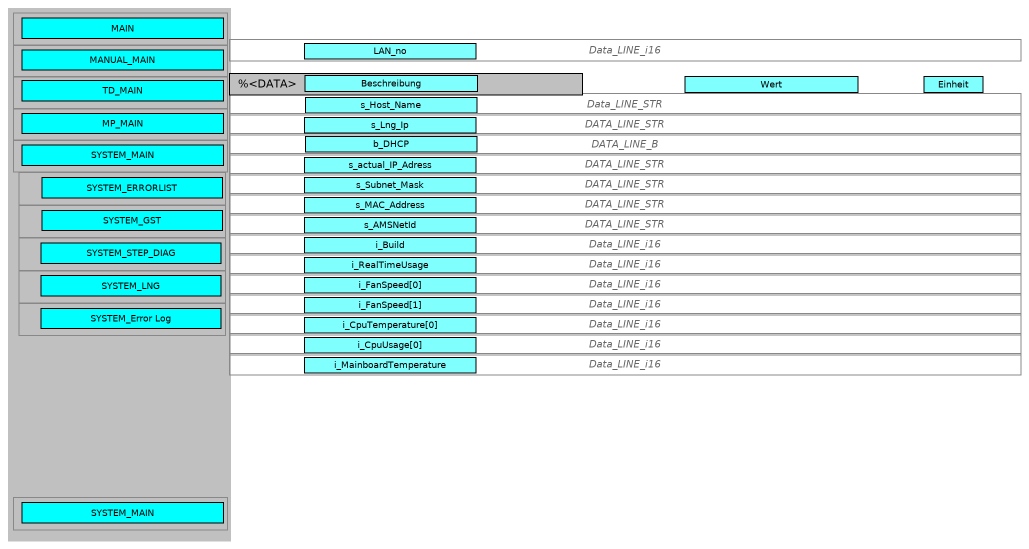
[picture p157: SYSTEM_MAIN (HMI screen)]
embedded screen at (3,115)-(226,648): M0003_System
embedded screen at (224,200)-(1016,222): Data_LINE_STR
embedded screen at (224,240)-(1016,262): DATA_LINE_B
rectangle at (300,204)-(472,220): text "s_Host_Name"; invisible if TRUE
rectangle at (300,243)-(472,259): text "b_DHCP"; invisible if TRUE
embedded screen at (224,260)-(1016,282): DATA_LINE_STR
rectangle at (299,264)-(471,280): text "s_actual_IP_Adress"; invisible if TRUE
embedded screen at (224,280)-(1016,302): DATA_LINE_STR
rectangle at (299,284)-(471,300): text "s_Subnet_Mask"; invisible if TRUE
embedded screen at (224,300)-(1016,322): DATA_LINE_STR
rectangle at (299,304)-(471,320): text "s_MAC_Address"; invisible if TRUE
embedded screen at (224,320)-(1016,342): DATA_LINE_STR
rectangle at (299,324)-(471,340): text "s_AMSNetId"; invisible if TRUE
embedded screen at (224,340)-(1016,362): Data_LINE_i16
rectangle at (299,344)-(471,360): text "i_Build"; invisible if TRUE
embedded screen at (224,360)-(1016,382): Data_LINE_i16
rectangle at (299,364)-(471,380): text "i_RealTimeUsage"; invisible if TRUE
embedded screen at (224,380)-(1016,402): Data_LINE_i16
rectangle at (299,384)-(471,400): text "i_FanSpeed[0]"; invisible if TRUE
embedded screen at (224,400)-(1016,422): Data_LINE_i16
rectangle at (299,404)-(471,420): text "i_FanSpeed[1]"; invisible if TRUE
embedded screen at (224,420)-(1016,442): Data_LINE_i16
rectangle at (299,424)-(471,440): text "i_CpuTemperature[0]"; invisible if TRUE
embedded screen at (224,440)-(1016,462): Data_LINE_i16
rectangle at (299,444)-(471,460): text "i_CpuUsage[0]"; invisible if TRUE
embedded screen at (224,460)-(1016,482): Data_LINE_i16
rectangle at (299,464)-(471,480): text "i_MainboardTemperature"; invisible if TRUE
embedded screen at (224,180)-(978,202): DATA_HEADER
embedded screen at (224,220)-(1016,242): DATA_LINE_STR
rectangle at (299,224)-(471,240): text "s_Lng_Ip"; invisible if TRUE
embedded screen at (224,146)-(1016,168): Data_LINE_i16
rectangle at (299,150)-(471,166): text "LAN_no"; invisible if TRUE
*)

(* Visualisation 04_System/SYSTEM_STEP_DIAG
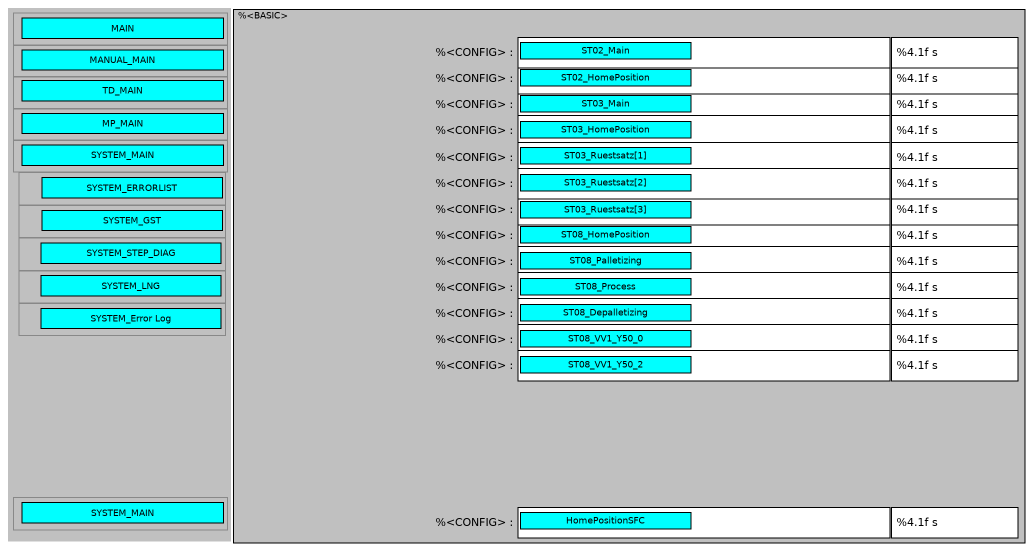
rectangle at (228,115)-(1020,649): text "%<BASIC>"; shows 'Prozess-Schrittketten'
embedded screen at (3,114)-(226,647): M0003_System
embedded screen at (282,195)-(1013,226): ZLIB_SFC_STATE
embedded screen at (282,221)-(1013,252): ZLIB_SFC_STATE
embedded screen at (282,326)-(1013,357): ZLIB_SFC_STATE
embedded screen at (282,352)-(1013,383): ZLIB_SFC_STATE
embedded screen at (282,378)-(1013,409): ZLIB_SFC_STATE
embedded screen at (282,404)-(1013,435): ZLIB_SFC_STATE
embedded screen at (282,430)-(1013,461): ZLIB_SFC_STATE
embedded screen at (282,456)-(1013,487): ZLIB_SFC_STATE
embedded screen at (282,300)-(1013,331): ZLIB_SFC_STATE
embedded screen at (282,613)-(1013,644): ZLIB_SFC_STATE
embedded screen at (282,169)-(1013,200): ZLIB_SFC_STATE
embedded screen at (282,143)-(1013,174): ZLIB_SFC_STATE
rectangle at (515,148)-(686,165): text "ST02_Main"; invisible if TRUE
rectangle at (515,175)-(686,192): text "ST02_HomePosition"; invisible if TRUE
rectangle at (515,201)-(686,218): text "ST03_Main"; invisible if TRUE
rectangle at (515,227)-(686,244): text "ST03_HomePosition"; invisible if TRUE
rectangle at (515,332)-(686,349): text "ST08_HomePosition"; invisible if TRUE
rectangle at (515,358)-(686,375): text "ST08_Palletizing"; invisible if TRUE
rectangle at (515,384)-(686,401): text "ST08_Process"; invisible if TRUE
rectangle at (515,410)-(686,427): text "ST08_Depalletizing"; invisible if TRUE
rectangle at (515,436)-(686,453): text "ST08_VV1_Y50_0"; invisible if TRUE
rectangle at (515,462)-(686,479): text "ST08_VV1_Y50_2"; invisible if TRUE
rectangle at (515,307)-(686,324): text "ST03_Ruestsatz[3]"; invisible if TRUE
rectangle at (515,618)-(686,635): text "HomePositionSFC"; invisible if TRUE
embedded screen at (282,248)-(1013,279): ZLIB_SFC_STATE
embedded screen at (282,274)-(1013,305): ZLIB_SFC_STATE
rectangle at (515,253)-(686,270): text "ST03_Ruestsatz[1]"; invisible if TRUE
rectangle at (515,280)-(686,297): text "ST03_Ruestsatz[2]"; invisible if TRUE
*)

(* Visualisation 02_TypeData/TD_01_EDIT
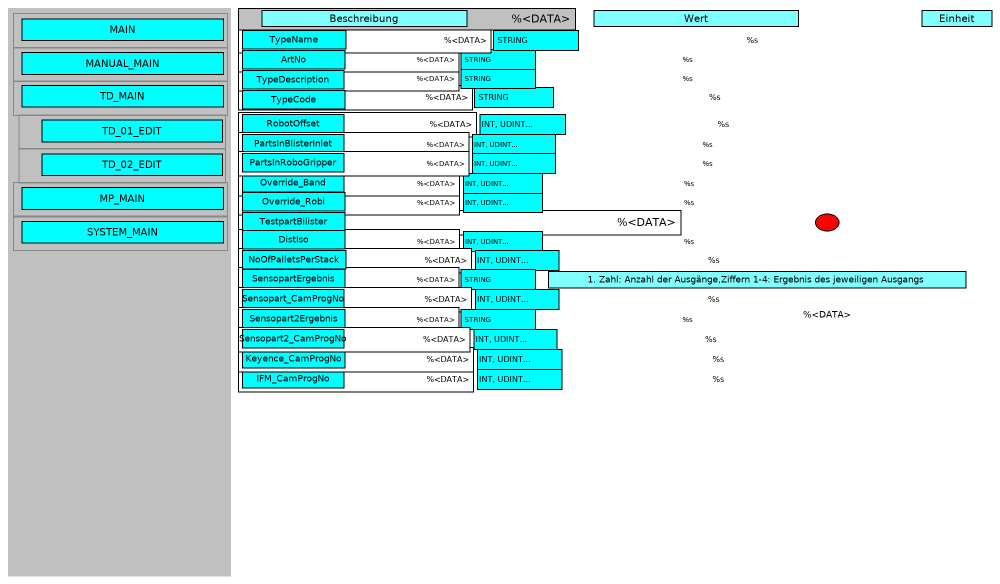
embedded screen at (3,115)-(226,683): M0003_TD
rectangle at (796,407)-(1009,436): text "%<DATA>"; shows 'Info_01'; invisible if gTypeCode<>4991 AND gTypeCode <>312
embedded screen at (233,317)-(834,342): Data_BOOL
embedded screen at (233,192)-(870,217): Data_STRING
embedded screen at (233,297)-(834,322): Data_DEZIMAL
embedded screen at (233,278)-(834,303): Data_DEZIMAL
embedded screen at (233,173)-(834,198): Data_STRING
embedded screen at (233,154)-(834,179): Data_STRING
embedded screen at (233,135)-(921,160): Data_STRING
embedded screen at (233,336)-(834,361): Data_DEZIMAL
embedded screen at (233,355)-(866,380): Data_DEZIMAL
embedded screen at (233,374)-(834,399): Data_STRING
rectangle at (237,137)-(341,156): text "TypeName"; invisible if TRUE
rectangle at (237,157)-(340,176): text "ArtNo"; invisible if TRUE
rectangle at (237,177)-(339,196): text "TypeDescription"; invisible if TRUE
rectangle at (237,197)-(340,216): text "TypeCode"; invisible if TRUE
rectangle at (237,280)-(339,299): text "Override_Band"; invisible if TRUE
rectangle at (237,299)-(340,318): text "Override_Robi"; invisible if TRUE
rectangle at (237,319)-(340,338): text "TestpartBilister"; invisible if TRUE
rectangle at (237,337)-(340,356): text "DistIso"; invisible if TRUE
rectangle at (237,376)-(340,395): text "SensopartErgebnis"; invisible if TRUE
rectangle at (237,357)-(341,376): text "NoOfPalletsPerStack"; invisible if TRUE
rectangle at (543,378)-(961,395): text "1. Zahl: Anzahl der Ausgänge,Ziffern 1-4: Ergebnis des jeweiligen Ausgangs"; invisible if TRUE
embedded screen at (233,219)-(879,244): Data_DEZIMAL
rectangle at (237,221)-(339,240): text "RobotOffset"; invisible if TRUE
embedded screen at (233,239)-(859,264): Data_DEZIMAL
rectangle at (237,241)-(339,260): text "PartsInBlisterInlet"; invisible if TRUE
embedded screen at (233,474)-(872,499): Data_DEZIMAL
rectangle at (237,476)-(339,495): text "IFM_CamProgNo"; invisible if TRUE
embedded screen at (233,394)-(866,419): Data_DEZIMAL
rectangle at (237,396)-(339,415): text "Sensopart_CamProgNo"; invisible if TRUE
embedded screen at (233,258)-(859,283): Data_DEZIMAL
rectangle at (237,260)-(339,279): text "PartsInRoboGripper"; invisible if TRUE
embedded screen at (233,115)-(987,137): DATA_HEADER_BEER
embedded screen at (233,454)-(872,479): Data_DEZIMAL
rectangle at (237,456)-(340,475): text "Keyence_CamProgNo"; invisible if TRUE
embedded screen at (233,414)-(834,439): Data_STRING
rectangle at (237,416)-(340,435): text "Sensopart2Ergebnis"; invisible if TRUE
embedded screen at (233,434)-(862,459): Data_DEZIMAL
rectangle at (237,436)-(339,455): text "Sensopart2_CamProgNo"; invisible if TRUE
*)

(* Visualisation 02_TypeData/TD_02_EDIT
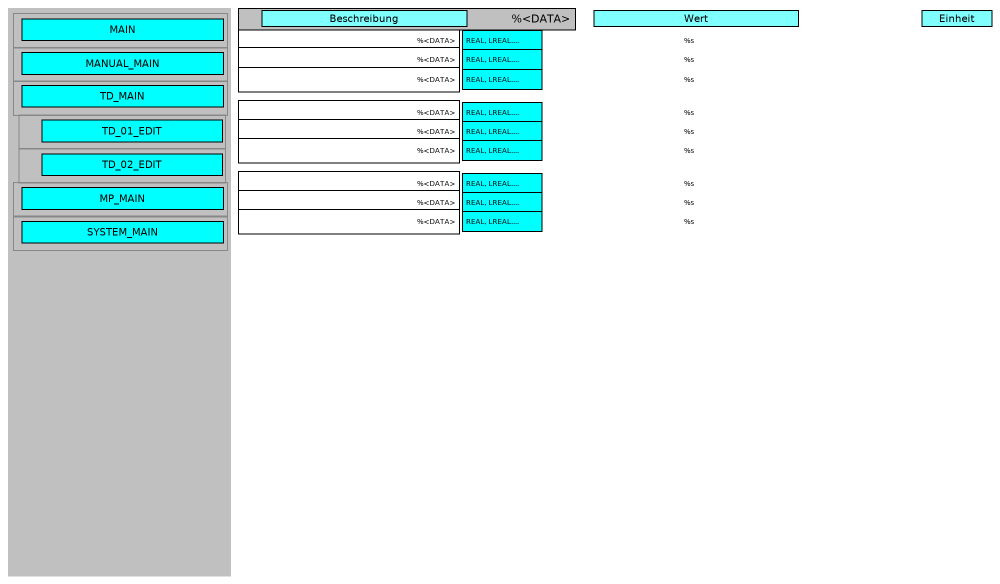
embedded screen at (3,115)-(226,683): M0003_TD
embedded screen at (233,135)-(834,160): Data_DEZIMAL_REAL
embedded screen at (233,154)-(834,179): Data_DEZIMAL_REAL
embedded screen at (233,174)-(834,199): Data_DEZIMAL_REAL
embedded screen at (233,207)-(834,232): Data_DEZIMAL_REAL
embedded screen at (233,226)-(834,251): Data_DEZIMAL_REAL
embedded screen at (233,245)-(834,270): Data_DEZIMAL_REAL
embedded screen at (233,115)-(987,137): DATA_HEADER_BEER
embedded screen at (233,278)-(834,303): Data_DEZIMAL_REAL
embedded screen at (233,297)-(834,322): Data_DEZIMAL_REAL
embedded screen at (233,316)-(834,341): Data_DEZIMAL_REAL
*)

(* Visualisation 02_TypeData/TD_MAIN
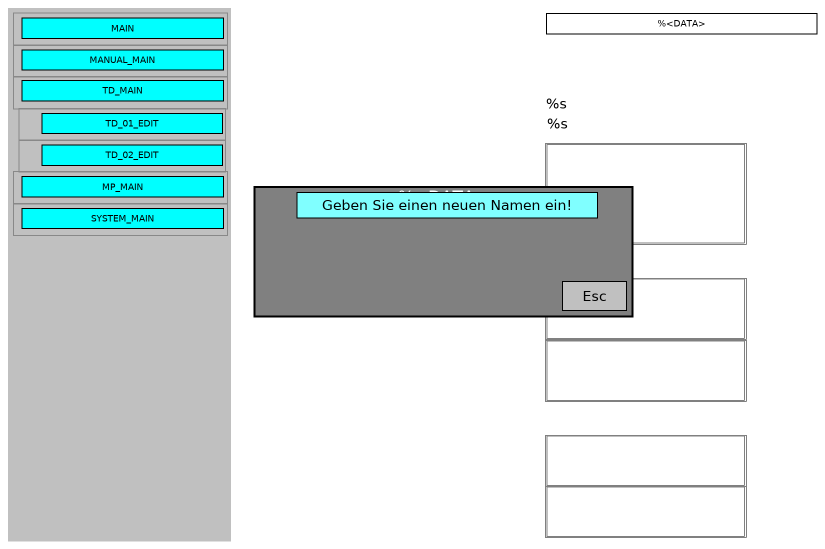
rectangle at (541,120)-(812,141): text "%<DATA>"; shows 'Filter'
embedded screen at (540,250)-(741,351): ZLIB_VISUBUTTON
embedded screen at (540,447)-(741,508): ZLIB_VISUBUTTON
embedded screen at (3,115)-(226,648): M0003_TD
embedded screen at (540,542)-(741,593): ZLIB_VISUBUTTON
embedded screen at (540,593)-(741,644): ZLIB_VISUBUTTON
embedded screen at (540,385)-(741,446): ZLIB_VISUBUTTON
embedded screen at (247,293)-(628,424): DIALOG_SAVE_AS
rectangle at (539,200)-(730,221): text "%s"; shows TDHandler.s_Typecode
rectangle at (540,220)-(731,241): text "%s"; shows TDHandler.s_Typedescription
2 elements of other kinds (tables, trends, ...) not read
*)

(* Visualisation zLibrary/ept/TEILEZAEHLER
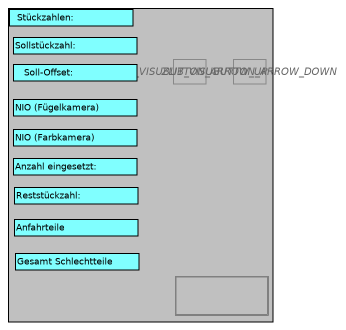
rectangle at (0,0)-(265,314): text "%<DATA>"; shows 'Parts'
rectangle at (10,23)-(157,48): text "%<DATA>"; shows 'PartsToProduce'
rectangle at (10,51)-(157,76): text "%<DATA>"; shows 'PartsToProduceOffset'
rectangle at (10,146)-(157,171): text "%<DATA>"; shows 'gPartsInserted'
rectangle at (10,176)-(157,201): text "%<DATA>"; shows 'PartsRemaining'
embedded screen at (165,51)-(198,76): ZLIB_VISUBUTTON_ARROW_UP
embedded screen at (225,51)-(258,76): ZLIB_VISUBUTTON_ARROW_DOWN
embedded screen at (167,268)-(260,307): ZLIB_VISUBUTTON_S18
rectangle at (10,116)-(157,141): text "%<DATA>"; shows 'gNokPartsColorCam'; invisible if gTypeCode<>5633 AND gTypeCode<>4991 AND gTypeCode <>312 AND gTypeCode <>322
rectangle at (10,86)-(157,111): text "%<DATA>"; shows 'gNokPartsWingCam'; invisible if gTypeCode<>4991 AND gTypeCode <>312
rectangle at (1,1)-(125,18): text "Stückzahlen:"; invisible if TRUE
rectangle at (5,29)-(129,46): text "Sollstückzahl:"; invisible if TRUE
rectangle at (5,56)-(129,73): text "Soll-Offset:"; invisible if TRUE
rectangle at (5,91)-(129,108): text "NIO (Fügelkamera)"; invisible if TRUE
rectangle at (5,121)-(129,138): text "NIO (Farbkamera)"; invisible if TRUE
rectangle at (5,150)-(129,167): text "Anzahl eingesetzt:"; invisible if TRUE
rectangle at (6,179)-(130,196): text "Reststückzahl:"; invisible if TRUE
rectangle at (10,207)-(166,232): text "%<DATA>"; shows 'Anfahrteile'
rectangle at (10,238)-(170,263): text "%<DATA>"; shows 'Gesamt Schlechtteile'
rectangle at (6,211)-(130,228): text "Anfahrteile"; invisible if TRUE
rectangle at (7,245)-(131,262): text "Gesamt Schlechtteile"; invisible if TRUE
9 elements of other kinds (tables, trends, ...) not read
*)

(* Visualisation zLibrary/MachineObjects/AnaIn/VANAIN
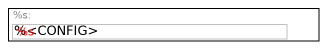
rectangle at (0,0)-(311,33): text "%s:"; shows $Object$.BitInName
rectangle at (0,12)-(281,33): text "%<CONFIG>"; shows $Object$.InstName
rectangle at (4,16)-(279,31): text "%s"; shows $Object$.ErrorString; invisible if NOT $Object$.ErrorPresent
1 elements of other kinds (tables, trends, ...) not read
*)

(* Visualisation zLibrary/MachineObjects/DigInOut/VBTN_SMAL
1 elements of other kinds (tables, trends, ...) not read
*)

(* Visualisation zLibrary/MachineObjects/DigIn/VDIGIN
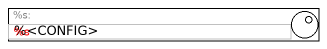
rectangle at (0,0)-(311,33): text "%s:"; shows $Object$.BitInName
rectangle at (0,12)-(281,33): text "%<CONFIG>"; shows $Object$.InstName
rectangle at (0,16)-(283,31): text "%s"; shows $Object$.ErrorString; invisible if NOT $Object$.ErrorPresent OR TRUE; alarm colour if $Object$.ErrorPresent
group at (283,3)-(310,30)
  ellipse at (0,0)-(27,27): alarm colour if $Object$.BitInToCheck; tooltip $Object$
  ellipse at (14,5)-(21,12): invisible if NOT $Object$.BitInToCheck
*)

(* Visualisation zLibrary/MachineObjects/DigInOut/VDIGOUT
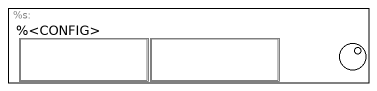
rectangle at (0,0)-(361,75): text "%s:"; shows $Object$.InstName
rectangle at (2,12)-(361,33): text "%<CONFIG>"; shows $Object$.InstName
embedded screen at (142,30)-(271,73): ZLIB_VISUBUTTON
group at (331,35)-(358,62)
  ellipse at (0,0)-(27,27): alarm colour if $Object$.BitOutToSet
  ellipse at (15,4)-(22,11): invisible if NOT $Object$.BitOutToSet
embedded screen at (11,30)-(140,73): ZLIB_VISUBUTTON
*)

(* Visualisation zLibrary/MachineObjects/DigInOut/VDIGOUT_SMAL
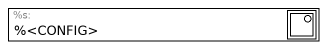
rectangle at (0,0)-(311,33): text "%s:"; shows $Object$.InstName; tooltip $Object$
rectangle at (0,12)-(311,33): text "%<CONFIG>"; shows $Object$.InstName; tooltip $Object$
rounded rectangle at (279,2)-(308,31): alarm colour if NOT $Object$.BtnOutput.Enable
rounded rectangle at (282,5)-(305,28): alarm colour if $Object$.BitOutToSet
ellipse at (296,7)-(303,14): invisible if NOT $Object$.BitOutToSet
2 elements of other kinds (tables, trends, ...) not read
*)

(* Visualisation zLibrary/MachineObjects/AnaIn/VENCODER
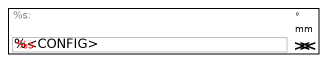
rectangle at (0,0)-(311,46): text "%s:"; shows $Object$.BitInName; alarm colour if $Object$.ErrorPresent
rectangle at (0,25)-(281,46): text "%<CONFIG>"; shows $Object$.InstName
rectangle at (4,29)-(279,44): text "%s"; shows $Object$.ErrorString; invisible if NOT $Object$.ErrorPresent OR TRUE
rectangle at (282,1)-(311,15): text "°"
rectangle at (282,14)-(311,28): text "mm"; invisible if $Object$.sInit.lr_LaengeProRpm = 0
rectangle at (282,25)-(312,50): text ">"; invisible if $Object$.Drehrichtung <> 1
rectangle at (282,25)-(312,50): text "<"; invisible if $Object$.Drehrichtung <> -1
rectangle at (282,25)-(312,50): text "><"; invisible if $Object$.Drehrichtung <> 0; alarm colour if $Object$.Reset; taps $Object$.Reset
2 elements of other kinds (tables, trends, ...) not read
*)

(* Visualisation zLibrary/VisuObjects/VISUBUTTON_TREE
1 elements of other kinds (tables, trends, ...) not read
*)

(* Visualisation zLibrary/X_MachSpec/ConveyorPartsIn/WPC_CONVEYOR_IN
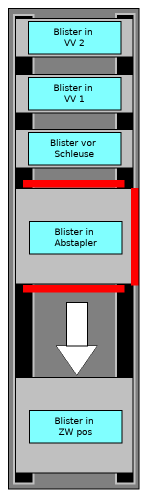
embedded screen at (48,294)-(89,367): SIGNS_ARROWDOWN
rectangle at (7,180)-(125,276): text "%<BASIC>"; shows 'Blister in Abstapler'; alarm colour if NOT ST08_404_B52_2.BitInToCheck; opens Visu.MainMenue.BtnManual_ST08_2.zoom
rectangle at (7,369)-(125,465): text "%<BASIC>"; shows 'Blister in ZW pos'; alarm colour if NOT ST08_406_B54_0.BitInToCheck; opens Visu.MainMenue.BtnManual_ST08_3.zoom
rectangle at (7,121)-(125,160): text "%<BASIC>"; shows 'Blister vor Schleuse'; alarm colour if NOT ST08_402_B51_2.BitInToCheck; opens Visu.MainMenue.BtnManual_ST08_1.zoom
rectangle at (7,66)-(125,105): text "%<BASIC>"; shows 'Blister in VV1'; invisible if NOT .MP.ST08.Trayzufuhr_Verlaengerung; alarm colour if NOT ST08_401_B50_5.BitInToCheck; opens Visu.MainMenue.BtnManual_ST08_1.zoom
rectangle at (7,10)-(125,49): text "%<BASIC>"; shows 'Blister in VV2'; invisible if NOT .MP.ST08.Trayzufuhr_Verlaengerung; alarm colour if NOT ST08_400_B50_0.BitInToCheck; opens Visu.MainMenue.BtnManual_ST08_1.zoom
rectangle at (20,13)-(113,46): text "Blister in / VV 2"; invisible if TRUE
rectangle at (20,69)-(113,102): text "Blister in / VV 1"; invisible if TRUE
rectangle at (20,124)-(113,157): text "Blister vor / Schleuse"; invisible if TRUE
rectangle at (21,213)-(114,246): text "Blister in / Abstapler"; invisible if TRUE
rectangle at (21,402)-(114,435): text "Blister in / ZW pos"; invisible if TRUE
embedded screen at (123,180)-(130,277): DOOR_LOCK
embedded screen at (15,172)-(116,179): DOOR_LOCK
embedded screen at (15,277)-(116,284): DOOR_LOCK
3 more shapes without text or variables
*)

(* Visualisation zLibrary/X_MachSpec/ConveyorPartsOut/WPC_CONVEYOR_OUT
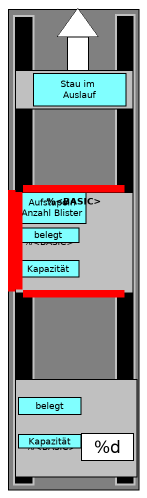
embedded screen at (49,-1)-(90,72): Signs_ArrowUp
rectangle at (7,61)-(125,100): text "%<BASIC>"; shows 'Stau im Auslauf'; alarm colour if NOT ST08_409_B55_5.BitInToCheck
rectangle at (25,64)-(118,97): text "Stau im / Auslauf"; invisible if TRUE
embedded screen at (7,370)-(129,468): WPC_OUT
embedded screen at (7,183)-(125,284): WPC_OUT_AUFSTAPELN
embedded screen at (7,183)-(14,280): DOOR_LOCK
embedded screen at (15,176)-(116,183): DOOR_LOCK
embedded screen at (15,281)-(116,288): DOOR_LOCK
embedded screen at (0,181)-(7,282): DOOR_LOCK
3 more shapes without text or variables
*)

(* Visualisation zLibrary/X_MachSpec/ConveyorPartsOut/WPC_OUT
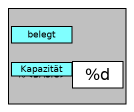
rectangle at (0,0)-(118,96): alarm colour if NOT ST08_406_B54_3.BitInToCheck OR ST08_406_B54_4.ValveSensor
rectangle at (2,16)-(64,43): text "%<BASIC>"; shows 'belegt'
rectangle at (64,53)-(115,80): text "%d"; shows TD.PartsInBlisterInlet
rectangle at (2,53)-(64,80): text "%<BASIC>"; shows 'Kapazität'
rectangle at (3,18)-(64,35): text "belegt"; invisible if TRUE
rectangle at (3,54)-(64,68): text "Kapazität"; invisible if TRUE
3 elements of other kinds (tables, trends, ...) not read
*)

(* Visualisation zLibrary/X_MachSpec/ConveyorPartsOut/WPC_OUT_AUFSTAPELN
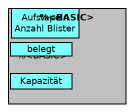
rectangle at (0,0)-(118,96): alarm colour if NOT ST08_407_B55_4.BitInToCheck
rectangle at (2,34)-(64,61): text "%<BASIC>"; shows 'belegt'
rectangle at (2,65)-(64,92): text "%<BASIC>"; shows 'Kapazität'
rectangle at (2,34)-(64,48): text "belegt"; invisible if TRUE
rectangle at (2,65)-(64,81): text "Kapazität"; invisible if TRUE
rectangle at (3,0)-(71,30): text "Aufstapeln / Anzahl Blister"; invisible if TRUE
rectangle at (0,3)-(118,31): text "%<BASIC>"; shows 'Aufstapeln Anzahl Blister'
3 elements of other kinds (tables, trends, ...) not read
*)

(* Visualisation zLibrary/ept/Axis/ZLIB_7211_ACHSE
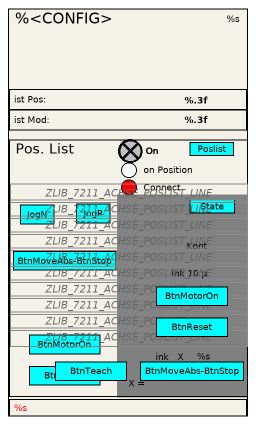
embedded screen at (0,0)-(241,408): ZLIB_7211_Control
embedded screen at (1,131)-(240,388): ZLIB_7211_ACHSE_Poslist
*)

(* Visualisation zLibrary/ept/Axis/ZLIB_7211_ACHSE_POSLIST
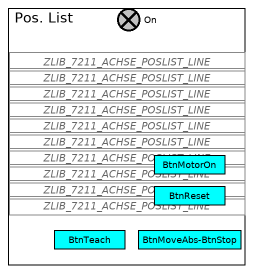
rectangle at (0,0)-(237,257): text "Pos. List"
embedded screen at (1,44)-(237,63): ZLIB_7211_ACHSE_POSLIST_LINE
embedded screen at (1,60)-(237,79): ZLIB_7211_ACHSE_POSLIST_LINE
embedded screen at (1,76)-(237,95): ZLIB_7211_ACHSE_POSLIST_LINE
embedded screen at (1,92)-(237,111): ZLIB_7211_ACHSE_POSLIST_LINE
embedded screen at (1,108)-(237,127): ZLIB_7211_ACHSE_POSLIST_LINE
embedded screen at (1,124)-(237,143): ZLIB_7211_ACHSE_POSLIST_LINE
embedded screen at (1,140)-(237,159): ZLIB_7211_ACHSE_POSLIST_LINE
embedded screen at (1,156)-(237,175): ZLIB_7211_ACHSE_POSLIST_LINE
embedded screen at (1,172)-(237,191): ZLIB_7211_ACHSE_POSLIST_LINE
embedded screen at (1,188)-(237,207): ZLIB_7211_ACHSE_POSLIST_LINE
rectangle at (130,222)-(233,241): text "BtnMoveAbs-BtnStop"; invisible if TRUE
rectangle at (46,222)-(117,241): text "BtnTeach"; invisible if TRUE
rounded rectangle at (134,1)-(237,22): text "On"
embedded screen at (109,0)-(132,23): SIGNS_Axis
rectangle at (146,147)-(217,166): text "BtnMotorOn"; invisible if TRUE
rectangle at (146,178)-(217,197): text "BtnReset"; invisible if TRUE
11 elements of other kinds (tables, trends, ...) not read
*)

(* Visualisation zLibrary/ept/Axis/ZLIB_7211_ACHSE_POSLIST_LINE
6 elements of other kinds (tables, trends, ...) not read
*)

(* Visualisation zLibrary/ept/Axis/ZLIB_7211_CONTROL
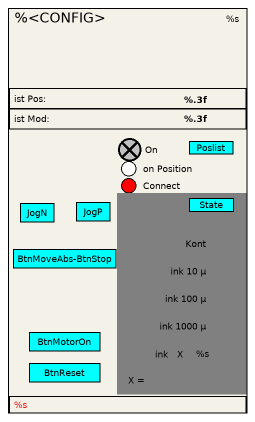
rectangle at (0,0)-(239,405): text "%<CONFIG>"; shows $Object$.sConfig.InstName
rectangle at (1,80)-(238,101): text "ist Pos:"; shows $Object$.sctrl.in.Position
rectangle at (1,100)-(238,121): text "ist Mod:"; shows $Object$.sPos.lr_Mod; invisible if NOT $Object$.sConfig.Modulo
rounded rectangle at (130,0)-(236,21): text "%s"; shows $Object$.sConfig.InstName
rectangle at (1,388)-(238,405): text "%s"; shows $Object$.LaufschriftObj.Display; invisible if $Object$.LaufschriftObj.Display=''
rounded rectangle at (135,131)-(238,152): text "On"
embedded screen at (110,130)-(133,153): SIGNS_Axis
ellipse at (113,153)-(128,168): alarm colour if $Object$.On_Position
rounded rectangle at (133,150)-(240,171): text "on Position"
ellipse at (113,170)-(128,185): alarm colour if $Object$.Connect
rounded rectangle at (133,167)-(240,188): text "Connect"
rectangle at (181,133)-(225,146): text "Poslist"; invisible if TRUE
embedded screen at (109,185)-(238,386): ZLIB_7211_STATE
embedded screen at (109,185)-(238,386): ZLIB_7211_OPT
rectangle at (68,194)-(102,213): text "JogP"; invisible if TRUE
rectangle at (12,195)-(46,214): text "JogN"; invisible if TRUE
rectangle at (21,324)-(92,343): text "BtnMotorOn"; invisible if TRUE
rectangle at (21,355)-(92,374): text "BtnReset"; invisible if TRUE
rectangle at (53,81)-(204,102): text "%.3f"; shows $Object$.sctrl.in.Position
rectangle at (53,100)-(204,121): text "%.3f"; shows $Object$.sPos.lr_Mod; invisible if NOT $Object$.sConfig.Modulo
rectangle at (5,241)-(108,260): text "BtnMoveAbs-BtnStop"; invisible if TRUE
20 elements of other kinds (tables, trends, ...) not read
*)

(* Visualisation zLibrary/ept/Axis/ZLIB_7211_OPT
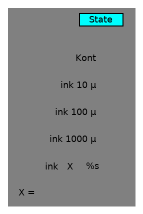
rectangle at (0,0)-(127,198): invisible if TRUE
rectangle at (27,42)-(93,58): text "Kont"; toggles $Object$.sVisuAxis.b_kont
rectangle at (27,69)-(93,85): text "ink 10 µ"; toggles $Object$.sVisuAxis.b_ink_10
rectangle at (26,96)-(93,112): text "ink 100 µ"; toggles $Object$.sVisuAxis.b_ink_100
rectangle at (26,123)-(93,139): text "ink 1000 µ"; toggles $Object$.sVisuAxis.b_ink_1000
rectangle at (32,151)-(70,166): text "ink   X"; toggles $Object$.sVisuAxis.b_ink_var
rectangle at (75,150)-(94,166): text "%s"; shows $Object$.sVisuAxis.Einheit_Pos; toggles $Object$.sVisuAxis.b_ink_var
rectangle at (5,177)-(32,192): text "X ="; toggles $Object$.sVisuAxis.b_ink_var
rectangle at (71,5)-(115,18): text "State"; invisible if TRUE
13 elements of other kinds (tables, trends, ...) not read
*)

(* Visualisation zLibrary/ept/Axis/ZLIB_7211_STATE
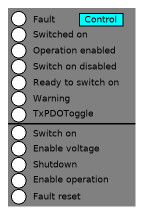
rectangle at (0,0)-(127,198): invisible if TRUE
ellipse at (3,67)-(18,82): alarm colour if $Object$.sCtrl.in.Ready_to_switch_on
rounded rectangle at (23,1)-(130,22): text "Fault"
ellipse at (3,19)-(18,34): alarm colour if $Object$.sCtrl.in.Switched_on
rounded rectangle at (23,16)-(130,37): text "Switched on"
ellipse at (3,35)-(18,50): alarm colour if $Object$.sCtrl.in.Operation_enabled
rounded rectangle at (23,32)-(130,53): text "Operation enabled"
ellipse at (3,3)-(18,18): alarm colour if $Object$.sCtrl.in.Fault
rounded rectangle at (23,64)-(130,85): text "Ready to switch on"
ellipse at (3,51)-(18,66): alarm colour if $Object$.sCtrl.in.Switch_on_disabled
rounded rectangle at (23,48)-(130,69): text "Switch on disabled"
ellipse at (3,83)-(18,98): alarm colour if $Object$.sCtrl.in.Warning
rounded rectangle at (23,80)-(130,101): text "Warning"
ellipse at (3,99)-(18,114): alarm colour if $Object$.sCtrl.in.TxPDOToggle
rounded rectangle at (23,95)-(130,116): text "TxPDOToggle"
ellipse at (3,117)-(18,132): alarm colour if $Object$.sCtrl.out.Switch_on
rounded rectangle at (23,115)-(130,136): text "Switch on"
ellipse at (3,133)-(18,148): alarm colour if $Object$.sCtrl.out.Enable_voltage
rounded rectangle at (23,130)-(130,151): text "Enable voltage"
ellipse at (3,149)-(18,164): alarm colour if $Object$.sCtrl.out.Shutdown
rounded rectangle at (23,146)-(130,167): text "Shutdown"
ellipse at (3,165)-(18,180): alarm colour if $Object$.sCtrl.out.Enable_operation
rounded rectangle at (23,161)-(130,182): text "Enable operation"
ellipse at (3,181)-(18,196): alarm colour if $Object$.sCtrl.out.Fault_reset
rounded rectangle at (23,178)-(130,199): text "Fault reset"
rectangle at (71,5)-(115,18): text "Control"; invisible if TRUE
1 more shapes without text or variables
1 elements of other kinds (tables, trends, ...) not read
*)

(* Visualisation zLibrary/MachineObjects/AnaIn/ZLIB_ANA_IN
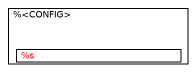
rectangle at (0,0)-(180,56): text "%<CONFIG>"; shows $Object$.InstName
rectangle at (8,41)-(173,54): text "%s"; shows $Object$.ErrorString; invisible if $Object$.ErrorString=''
2 elements of other kinds (tables, trends, ...) not read
*)

(* Visualisation zLibrary/MachineObjects/DigIn/ZLIB_DIG_IN
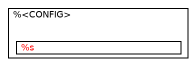
rectangle at (0,0)-(180,50): text "%<CONFIG>"; shows $Object$.InstName
rectangle at (8,33)-(173,46): text "%s"; shows $Object$.ErrorString; invisible if NOT $Object$.ErrorPresent
1 elements of other kinds (tables, trends, ...) not read
*)

(* Visualisation zLibrary/MachineObjects/DigInOut/ZLIB_DIGOUT
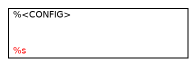
rectangle at (0,0)-(180,50): text "%<CONFIG>"; shows $Object$.InstName; alarm colour if $Object$.BitOutToSet
rounded rectangle at (0,36)-(177,50): text "%s"; shows $Object$.ErrorString; invisible if NOT $Object$.ErrorPresent
2 elements of other kinds (tables, trends, ...) not read
*)

(* Visualisation zLibrary/MachineObjects/DigInOut/ZLIB_DIGOUTIN
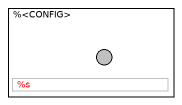
rectangle at (0,0)-(166,89): text "%<CONFIG>"; shows $Object$.InstName
rounded rectangle at (4,70)-(160,83): text "%s"; shows $Object$.ErrorString; invisible if NOT $Object$.ErrorPresent
ellipse at (88,41)-(104,57): invisible if NOT($Object$.BtnOutput.Visible); alarm colour if $Object$.BitOutToSet
3 elements of other kinds (tables, trends, ...) not read
*)

(* Visualisation zLibrary/MachineObjects/AnaIn/ZLIB_ENCODER_IN
